PROGRAM MAIN
VAR
	foo:INT;
END_VAR

END_PROGRAM

(* stored: Version 1.1.0.1, ProductVersion 3.1.4024.12
   POU MAIN: Id {5632992b-1cd1-4503-aa45-a8c114883fd6}, SpecialFunc None *)
